ABB RobotStudio station: SOCKET.rspag

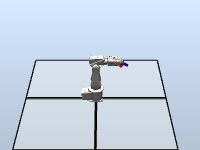
--- station ---
Station Station (saved by RobotStudio 6.8.8148.134)
Controller SOCKET
  mechanical unit ROB_1: IRB120_3_58__01, 6 joints, base frame (0, 0, 0) mm
Layout (positions relative to the parent item):
  - IRB120_3_58__01 [mechanism, from Robots\IRB120_3_58_G_01.rslib] at (0, 0, 0) mm; joint values [0, 0, 0, 0, 0.5236, 0] (rad or m)

--- Backups/SOCKET/RAPID/TASK1/PROGMOD/Module1.mod ---
MODULE Module1
VAR socketdev Socket_Lmsa;
VAR socketdev Socket1;
VAR string str;
VAR byte rec{50};
VAR byte send{50};

    PROC outsend()
        SocketClose Socket_Lmsa;
        SocketCreate Socket_Lmsa;
        SocketConnect Socket_Lmsa,"192.168.110.124",2000;
        SocketSend Socket_Lmsa\Data:=send;
        !SocketSend Socket_Lmsa\str:=str;
        SocketClose Socket_Lmsa;
    ENDPROC


    PROC intrec()
        SocketClose Socket_Lmsa;
        SocketCreate Socket_Lmsa;
        SocketConnect Socket_Lmsa,"192.168.110.124",2000;

        SocketReceive Socket_Lmsa\Data:=rec;

        !SocketReceive Socket_Lmsa\Str:=str;
        SocketClose Socket_Lmsa;
    ENDPROC



    PROC socke01()
        SocketCreate Socket1;
        !SocketConnect Socket1,"127.0.0.1",2000;
        SocketConnect Socket1,"192.168.110.123",2000;
        WHILE TRUE DO
            SocketSend Socket1\str:="hello socket";
            SocketReceive Socket1\Str:=str;
            TPWrite"socket:"+str;
        ENDWHILE
     ENDPROC

    PROC main()
        FOR i FROM 11 TO 60 DO
           send{i-10}:=i;
        ENDFOR
     !   server;
    !    socke01;
      intrec;
      !outsend;


     ENDPROC
     PROC server()
        SocketCreate Socket1;
        SocketBind Socket1,"192.168.110.123",2000;
        SocketListen Socket1;
        SocketAccept Socket1, Socket_Lmsa;
        WHILE TRUE DO
            !SocketReceive Socket_Lmsa\Str:=str;
            !TPWrite"socket:"+str;
            SocketSend Socket_Lmsa\Data:=send;
            WaitTime 1;
        ENDWHILE


    ENDPROC
ENDMODULE

--- Backups/SOCKET/SYSPAR/EIO.cfg ---
EIO:CFG_1.0:6:1::
#
INDUSTRIAL_NETWORK:

      -Name "DeviceNet" -Label "DeviceNet Master/Slave Network" -Address "2"

      -Name "PROFINET" -Connection "PROFINET Network"\
      -Label "PROFINET Controller/Device Network" -StationName ""
#
DEVICENET_DEVICE:

      -Name "d652" -VendorName "ABB Robotics" -ProductName "24 VDC I/O Device"\
      -Label "DSQC 652 24 VDC I/O Device" -ProductCode 26 -DeviceType 7\
      -ConnectionType "COS" -OutputSize 2 -InputSize 2
#
DEVICENET_INTERNAL_DEVICE:

      -Name "DN_Internal_Device" -VendorName "ABB Robotics"\
      -ProductName "DeviceNet Internal Slave Device"
#
PROFINET_DRIVER:

      -Name "PROFINET_COMMON_DATA"
#
PROFINET_INTERNAL_DEVICE:

      -Name "PN_Internal_Device" -VendorName "ABB Robotics"\
      -ProductName "PROFINET Internal Device"
